Xinje XDPPro project, PLC1: XDH-60T4 (software 3.7.18 2024-11-27)

PROGRAM 梯形图

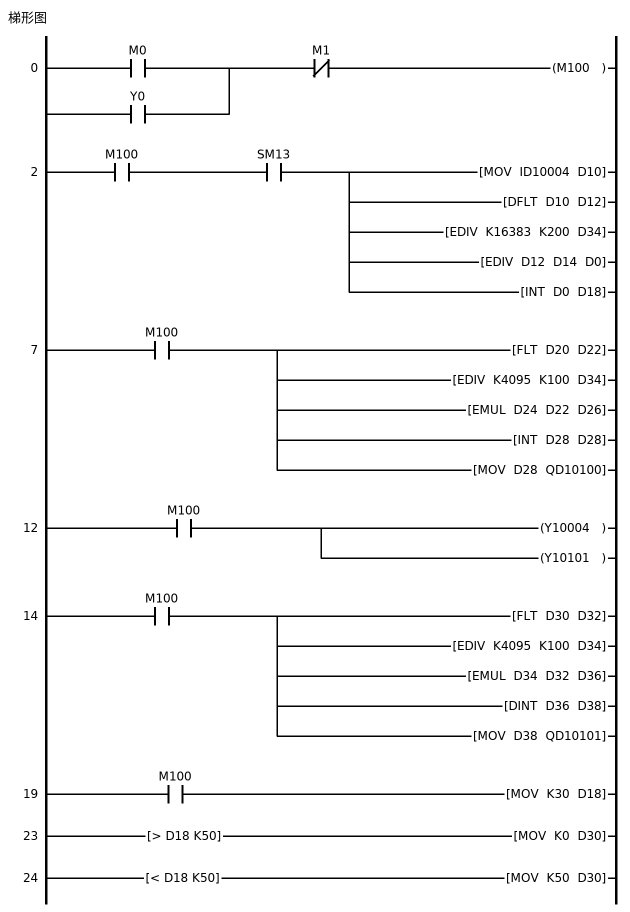
LD     M0
OR     Y0
ANI    M1
OUT    M100
LD     M100
AND    SM13
MOV    ID10004 D10
DFLT   D10 D12
EDIV   K16383 K200 D34
EDIV   D12 D14 D0
INT    D0 D18
LD     M100
FLT    D20 D22
EDIV   K4095 K100 D34
EMUL   D24 D22 D26
INT    D28 D28
MOV    D28 QD10100
LD     M100
OUT    Y10004
OUT    Y10101
LD     M100
FLT    D30 D32
EDIV   K4095 K100 D34
EMUL   D34 D32 D36
DINT   D36 D38
MOV    D38 QD10101
LD     M100
MOV    K30 D18
LD>    D18 K50
MOV    K0 D30
LD<    D18 K50
MOV    K50 D30